# B&R Automation Studio project perfxxl (part 10)

#### pro_v.c
```c
#ifdef _DEFAULT_INCLUDES
	#include <AsDefault.h>
#endif
/*
                             *******************
******************************* C SOURCE FILE *******************************
**                           *******************                           **
**                                                                         **
** project  : BlueFin                                                      **
** filename : PRO_V.C                                                      **
** version  : 1.01                                                         **
** date     : 16.10.2008                                                   **
**                                                                         **
*****************************************************************************
** Abstract                                                                **
** ========                                                                **
**                                                                         **
** Copyright (c) 2008, Krause-Biagosch GmbH                                **
** All rights reserved.                                                    **
**                                                                         **
*****************************************************************************
VERSION HISTORY:
----------------
Version     : 1.00
Date        : 14.10.2008
Revised by  : Herbert Aden
Description : Original version

Version     : 1.01
Date        : 16.10.2008
Revised by  : Herbert Aden
Description : Pumps now only active, if machine is in ON mode

*/
#define _PRO_V_C_SRC

/****************************************************************************/
/**                                                                        **/
/**                           INCLUDE FILES                                **/
/**                                                                        **/
/****************************************************************************/

#include "glob_var.h"
#include "egmglob_var.h"
#include <math.h>

/****************************************************************************/
/**                                                                        **/
/**                       DEFINITIONS AND MACROS                           **/
/**                                                                        **/
/****************************************************************************/
/* NONE */

/****************************************************************************/
/**                                                                        **/
/**                      TYPEDEFS AND STRUCTURES                           **/
/**                                                                        **/
/****************************************************************************/
/* NONE */

/****************************************************************************/
/**                                                                        **/
/**                      PROTOTYPES OF LOCAL FUNCTIONS                     **/
/**                                                                        **/
/****************************************************************************/
/* NONE */

/****************************************************************************/
/**                                                                        **/
/**                      EXPORTED VARIABLES                                **/
/**                                                                        **/
/****************************************************************************/
/* NONE */

/****************************************************************************/
/**                                                                        **/
/**                           GLOBAL VARIABLES                             **/
/**                                                                        **/
/****************************************************************************/
/***
***/

/****************************************************************************/
/**                                                                        **/
/**                      TASK-LOCAL VARIABLES                              **/
/**                                                                        **/
/****************************************************************************/
_LOCAL    INT                 RefillStep;

/****************************************************************************/
/**                                                                        **/
/**                    MODULE-LOCAL VARIABLES                              **/
/**                                                                        **/
/****************************************************************************/
static    TON_10ms_typ        ReplPumpTimer;
static    TON_10ms_typ        CanisterFullTimer;
static    TOF_10ms_typ        CanisterNotFullTimer;

/****************************************************************************/
/**                                                                        **/
/**                      EXTERNAL VARIABLES                                **/
/**                                                                        **/
/****************************************************************************/

/****************************************************************************/
/**                                                                        **/
/**                          EXPORTED FUNCTIONS                            **/
/**                                                                        **/
/****************************************************************************/

void InitProV(void)
{
	RefillStep = 0;
	CanisterFullTimer.IN    = FALSE;
	CanisterNotFullTimer.IN = FALSE;
	ReplPumpTimer.IN = FALSE;
}

void ProV(void)
{

/*
 * Umwälzung immer, solange nicht leer (Levelswitch ist scließer!)
 */
	Out_DevCanister_Circulation =  In_DevCanister_Empty
								&& ControlVoltageOk
								&& EGMDeveloperTank.Enable;

	CanisterFullTimer.IN    = In_DevCanister_Full;
	CanisterNotFullTimer.IN = In_DevCanister_Full;
	CanisterFullTimer.PT = 1000;
	CanisterNotFullTimer.PT = 1000;
	TON_10ms(&CanisterFullTimer);
	TOF_10ms(&CanisterNotFullTimer);

	TON_10ms(&ReplPumpTimer);
/*
 * Befüllpumpe an für 1 min, wenn Levelschalter "voll" weggeht
 * Wenn Schalter wiederkommt, dann auf jeden Fall aus
 */

	if( !ControlVoltageOk
 	 || !EGMDeveloperTank.Enable
 	 )
 	{
 		RefillStep = 0;
 		ReplPumpTimer.IN = FALSE;
		Out_DevCanister_Replenish = FALSE;
 	}

	switch (RefillStep)
	{
		case 0:
		{
			if( !ControlVoltageOk
		 	 || !EGMDeveloperTank.Enable
		 	 )
		 		break;

		/* Pumpe an, Wartezeit 0,5 min triggern*/
			if(!CanisterNotFullTimer.Q)
			{
				ReplPumpTimer.IN = TRUE;
				ReplPumpTimer.PT = EGMAutoParam.PROV_PumpOnTime;
				Out_DevCanister_Replenish = TRUE;
				RefillStep = 10;
				break;
			}

			break;
		}
		case 10:
		{
		/* Wartezeit abgelaufen: Pumpe aus,nächster Schritt*/
			if(ReplPumpTimer.Q)
			{
				Out_DevCanister_Replenish = FALSE;
				ReplPumpTimer.IN = FALSE;
				RefillStep = 20;
				break;
			}
		/* Kanister wieder voll: Pumpe aus und fertig*/
			if(CanisterFullTimer.Q)
			{
				ReplPumpTimer.IN = FALSE;
				RefillStep = 0;
				Out_DevCanister_Replenish = FALSE;
				break;
			}

			break;
		}
		case 20:
		{
		/* Warten eine min */
			if(ReplPumpTimer.Q)
			{
				ReplPumpTimer.IN = FALSE;
				RefillStep = 0;
				break;
			}
			ReplPumpTimer.IN = TRUE;
			ReplPumpTimer.PT = EGMAutoParam.PROV_PumpOffTime; /* 5 min */
			break;
		}
	}

}
```

### Program Logical/Processor/egmauto (ANSIC, version 0.00.0)

#### auto.c
```c
#ifdef _DEFAULT_INCLUDES
	#include <AsDefault.h>
#endif
/*************************************************************************************************
 Handling of Automatic mode

*************************************************************************************************/

/****	Bedeutung der Ampel Signale

o = AUS, X = AN, b = blinkt

					Grün		Gelb		Rot
Aus					o			o			X
Aufheizen			o			o			X
Betriebsbereit		X			o			o
Verarbeitung		o			X			o
Reinigung			o			b			o
Störung				o			o			b
***/

/*********************************************************************************/
/*	Alarmliste */
/**
x	EGM_AlarmBitField[0]	AlarmNr 1	Notaus
x	EGM_AlarmBitField[1]	AlarmNr 2	kein Antriebstakt
x	EGM_AlarmBitField[2]	AlarmNr 3	EGMGummierung Füllstand zu niedrig
x	EGM_AlarmBitField[3]	AlarmNr 4	Vorspülen Füllstand zu niedrig
x	EGM_AlarmBitField[4]	AlarmNr 5	Nachspülen Füllstand zu niedrig
x	EGM_AlarmBitField[5]	AlarmNr 6	Entwickler Füllstand zu niedrig
x	EGM_AlarmBitField[6]	AlarmNr 7	Entwickler Temperatur zu niedrig
x	EGM_AlarmBitField[7]	AlarmNr 8	Entwickler Temperatur zu hoch
x	EGM_AlarmBitField[8]	AlarmNr 9	Nacherwärmung 1 Temperatur zu niedrig
x	EGM_AlarmBitField[9]	AlarmNr 10	Nacherwärmung 1 Temperatur zu hoch
x	EGM_AlarmBitField[10]	AlarmNr 11	Nacherwärmung 2 Temperatur zu niedrig
x	EGM_AlarmBitField[11]	AlarmNr 12	Nacherwärmung 2 Temperatur zu hoch
x	EGM_AlarmBitField[12]	AlarmNr 13	Plattenstau
	EGM_AlarmBitField[13]	AlarmNr 14	Entwickler zu alt
	EGM_AlarmBitField[14]	AlarmNr 15	E/A Modul nicht gefunden
x	EGM_AlarmBitField[15]	AlarmNr 16	Nacherw. Sensor 1 defekt
x	EGM_AlarmBitField[16]	AlarmNr 17	Nacherw. Sensor 2 defekt
x	EGM_AlarmBitField[17]	AlarmNr 18	Nacherw. Umgeb. Sensor defekt
x	EGM_AlarmBitField[18]	AlarmNr 19	Entwickler Temp. Sensor defekt
x	EGM_AlarmBitField[19]	AlarmNr 20	Nacherw. Heizung 1 defekt
x	EGM_AlarmBitField[20]	AlarmNr 21	Nacherw. Heizung 2 defekt
	EGM_AlarmBitField[21]	AlarmNr 22	Vorspülstation Befüllen fehlgeschlagen
	EGM_AlarmBitField[22]	AlarmNr 23	Nachspülstation Befüllen fehlgeschlagen
	EGM_AlarmBitField[23]	AlarmNr 24	Entwickler Befüllen fehlgeschlagen
x	EGM_AlarmBitField[24]	AlarmNr 25	Nacherwärmung 1 überhitzt
x	EGM_AlarmBitField[25]	AlarmNr 26	Nacherwärmung 2 überhitzt
x	EGM_AlarmBitField[26]	AlarmNr 27	Entwickler überhitzt
x	EGM_AlarmBitField[27]	AlarmNr 28	Antrieb: Geschwindigkeitsabweichung zu groß
x	EGM_AlarmBitField[28]	AlarmNr 29	Temperaturmodul nicht gefunden
**/

#include "EGMglob_var.h"
#include "glob_var.h"
#include "auxfunc.h"

#define MM_PER_PULSE (251.0/18.0)
#define NUMBER_OF_TIMING_CYCLES 10

#define LAMPTESTTIME 50 /*  *10 ms*/

_GLOBAL BOOL	Clock_1s;

R_TRIGtyp	RPMSignalEdgeR;

R_TRIGtyp	InputSensorEdgeR,OutputSensorEdgeR;
F_TRIGtyp	InputSensorEdgeF,OutputSensorEdgeF;
TON_10ms_typ	PlateInputTimer,StandbyDelay;
TON_10ms_typ	InputSensorOnDelay,OutputSensorOnDelay,ProcessingTimer;
TOF_10ms_typ	InputSensorOffDelay,OutputSensorOffDelay;

/*Timer für Spülprogramm*/
TON_10ms_typ	CleaningTimer;

BOOL AutoInit,OffInit,WaitForStandby;
_GLOBAL REAL PlateLength; /* wird in lccount berechnet */
_LOCAL	STRING CurrentPlateName[MAXPLATETYPENAME+6];
_LOCAL	INT PlatesInMachine,TimeAtPlateInput;
_LOCAL INT	DontCheckHeating;
REAL tmpval;
int i;
BOOL	 EnablePulseCounter;
_LOCAL BOOL	OnButton,OffButton;
_LOCAL UDINT CleaningTimerDisplay,CleaningTimerOverallDisplay;

_LOCAL UDINT	TEST;

/* Variable, die genauso lange true ist, wie der sensor Eingang, aber über  ein- und ausschaltverzögerung entprellt*/
_GLOBAL	BOOL PlateOverSensor;

/* Variablen für Ampelansteuerung, interne Merker, werden an zentraler Stelle auf die Ausgänge kopiert
wegen Lampentest Funktion*/
BOOL	InternalLightGreen;
BOOL	InternalLightRed;
BOOL	InternalLightYellow;
BOOL	FatalError;
_LOCAL BOOL TriggerLampTest;
TON_10ms_typ		HornTimer1,HornTimer2,LampTestTimer;
int LampTestStep,LampTestCycle,LampTestReturnStep;
TP_10ms_typ		BlinkTimer1,BlinkTimer2;

F_TRIGtyp ServiceKeyEdgeF;

R_TRIGtyp AlarmTrigger[EGM_MAXALARMS];
_GLOBAL BOOL	HornActive;

static    TON_10ms_typ        WaitForOutputTimer;
static	BOOL	OutputBlocked;

/**
	Bei allen Platten im FIFO die Position um Betrag X erhöhen
**/
void FIFOChangePlatePosition(REAL X)
{
	int i = 0;
	REAL BackEnd;
	do
	{
		if (EGMPlateFIFO[i].Used)
		{
			EGMPlateFIFO[i].Position += X;
			BackEnd = (EGMPlateFIFO[i].Position - EGMPlateFIFO[i].Length);
			/* Trigger Waiting for output
			 */
			if(  (EGMPlateFIFO[i].Position > ((MACHINELENGTH - 0.35) * 1000))
			  && (EGMPlateFIFO[i].Status != PS_OUTPUTREACHED)
			  )
				EGMPlateFIFO[i].Status = PS_WAITINGFOROUTPUT;

			if(  (BackEnd > ((MACHINELENGTH + 0.15) * 1000))
			  && (EGMPlateFIFO[i].Status == PS_OUTPUTREACHED)
			  )
			{
				OutputBlocked = TRUE;
			}
		}
		i++;
	}
	while (i <FIFOLENGTH);

}

/**
	Alle Platten im FIFO um 1 Platz weiterrücken
**/
void FIFOShift(void)
{
	int i = FIFOLENGTH-2;

	do
	{
		if (EGMPlateFIFO[i].Used)
		{
			EGMPlateFIFO[i+1] = EGMPlateFIFO[i];
		}
		i--;
	}
	while (i>=0);
	EGMPlateFIFO[0].Used = FALSE;
	EGMPlateFIFO[0].Position = 0;
	EGMPlateFIFO[0].Length =  0;
	EGMPlateFIFO[0].Status = PS_NONE;
}

/**
	FIFO mit Platten für die Darstellung bearbeiten
**/
void HandleFIFO()
{
	RPMSignalEdgeR.CLK = RPMCheck;
	R_TRIG(&RPMSignalEdgeR);
	if ((CurrentMode == M_AUTO)
	&& ((CurrentState==S_PROCESSING) || (CurrentState==S_STARTPROCESSING))
	)
	{
/* mit jedem Antriebspuls werden die Platten um einen festen Betrag X weitergefördert*/
		if(RPMSignalEdgeR.Q )
			FIFOChangePlatePosition(MM_PER_PULSE);

/* mit steigender Flanke eine neue Platte im FIFO erzeugen*/
		if(InputSensorEdgeR.Q)
		{
			EGMPlateFIFO[0].Used = TRUE;
			EGMPlateFIFO[0].Position = 0;
			EGMPlateFIFO[0].Length =  0;
			EGMPlateFIFO[0].Status = PS_RUNNING;
		}
/*wenn im FIFO eine Platte am Anfang steht und der Sensor belegt bleibt, wird diese länger*/
		if(PlateOverSensor)
		{
			if(RPMSignalEdgeR.Q )
				EGMPlateFIFO[0].Length += MM_PER_PULSE;
		}
/* mit fallender Flanke die Platte im FIFO weiterschieben*/
		if(InputSensorEdgeF.Q)
		{
			FIFOShift();
			if(EGMPlatesInFIFO < (FIFOLENGTH - 1) )
				EGMPlatesInFIFO++;
		}

/* mit steigender Flanke des Ausgangssensors den Status der letzten Platte im FIFO wechseln */
		if(OutputSensorEdgeR.Q)
		{
			if (EGMPlatesInFIFO > 0 && EGMPlatesInFIFO < FIFOLENGTH)
			{
				if(EGMPlateFIFO[EGMPlatesInFIFO].Status == PS_WAITINGFOROUTPUT)
					EGMPlateFIFO[EGMPlatesInFIFO].Status = PS_OUTPUTREACHED;
			}
		}

/* mit fallender Flanke des Ausgangssensors die letzte Platte im FIFO Löschen*/
		if(OutputSensorEdgeF.Q)
		{
			if(OutputBlocked)
				EGM_AlarmBitField[12] = 0;

			OutputBlocked = FALSE;
			if (EGMPlatesInFIFO > 0 && EGMPlatesInFIFO < FIFOLENGTH)
			{
				EGMPlateFIFO[EGMPlatesInFIFO].Used = FALSE;
				EGMPlateFIFO[EGMPlatesInFIFO].Position = 0;
				EGMPlateFIFO[EGMPlatesInFIFO].Length =  0;
				EGMPlateFIFO[EGMPlatesInFIFO].Status = PS_NONE;
				EGMPlatesInFIFO--;
			}
		}
/* Auslauf blockiert: warten, bis alle Platten raus sind, dann Fehlermeldung*/
		if(OutputBlocked)
		{
			int i;
			REAL BackEnd;
			for(i=FIFOLENGTH;i>0;i--)
			{
				if(EGMPlateFIFO[i].Used)
				{
					BackEnd = (EGMPlateFIFO[i].Position - EGMPlateFIFO[i].Length);
					if(BackEnd > ((MACHINELENGTH - 0.35) * 1000))
					{
						EGMPlateFIFO[i].Used = FALSE;
						EGMPlateFIFO[i].Position = 0;
						EGMPlateFIFO[i].Length =  0;
						EGMPlateFIFO[i].Status = PS_NONE;
						if(EGMPlatesInFIFO > 0)
							EGMPlatesInFIFO--;
						if(PlatesInMachine > 0)
							PlatesInMachine--;
					}
				}
			}
			if(EGMPlatesInFIFO == 0 && !EGM_AlarmBitField[12])
			{
				ShowMessage(104,138,0,CAUTION,OKONLY, FALSE);
				EGM_AlarmBitField[12] = 1;
			}
		}

	}
	else
	if (((CurrentMode == M_AUTO)&& (CurrentState == S_READY))
	|| (PlatesInMachine == 0)
	)
	{
		int i;
		EGMPlatesInFIFO = 0;
		for( i = 0; i < FIFOLENGTH; i++)
		{
			EGMPlateFIFO[i].Used = 0;
			EGMPlateFIFO[i].Position = 0;
			EGMPlateFIFO[i].Length =  0;
		}
	}
}

int	FindPlateType(UDINT parLength)
{
	int i;
	int Deviation,MinDeviation,PosInTable;
	BOOL	transverse;

	MinDeviation = 32000; /* Startwert: Abweichung riesig*/
	transverse = FALSE;
	for (i=1;i<MAXPLATETYPES;i++)
	{
		Deviation = abs(EGMPlateTypes[i].SizeX - parLength);
		if (Deviation < MinDeviation)
		{
			MinDeviation = Deviation;
			PosInTable = i;
			transverse = FALSE;
		}
/*
		Deviation = abs(EGMPlateTypes[i].SizeY - parLength);
		if (Deviation < MinDeviation)
		{
			MinDeviation = Deviation;
			PosInTable = i;
			transverse = TRUE;
		}
*/
	}
	if (transverse)
		return PosInTable+MAXPLATETYPES;
	else
		return PosInTable;
}

void LampAndHorn(void)
{
	int i,j,k;
/*
 * definiert die Alarme, die eine Meldung auf dem Hauptbild auslösen
 * -1 ist Ende Kennung der Liste!
 * Achtung: Bei Veränderung muss auch in pics.c "case 101" angepasst werden
 *          Alarmnummern um 1 versetzt zu Alarmnummer in Visu, zB AlarmNr 49 zeigt
 *          in Visu Alarmnummer 50 an!!
 */
	int MessageAlarms[]={0,2,12,33,34,35,36,37,38,39,40,-1};

/* ********************************************************************************/
/* Ampel */
/* ********************************************************************************/
	BlinkTimer1.PT = 30;
	BlinkTimer2.PT = 30;
	TON_10ms(&LampTestTimer);
	BlinkTimer1.IN = ! BlinkTimer2.Q;
	TP_10ms(&BlinkTimer1);
	BlinkTimer2.IN = ! BlinkTimer1.Q;
	TP_10ms(&BlinkTimer2);

	switch (LampTestStep)
	{
		case 0:
		{
			int i;
			BOOL flag;
			flag = 0;
			for (i=0;i<EGM_MAXALARMS;i++)
			{
/* EGMPreheat Temperatur zu niedrig nur relevant, wenn der Regler auch an ist*/
				if (i==8 || i==10)
					flag = flag || (EGM_AlarmBitField[i] && EGMPreheat.Enable && !DontCheckHeating);
				else
					flag = flag || EGM_AlarmBitField[i];
			}

/*solange kein Lampentest ist: interne Ampelmerker auf Ausgänge kopieren*/
			if (flag)
			{
				LightRed = BlinkTimer1.Q;
				LightGreen = 0;
				LightYellow = 0;
			}
			else
			{
				LightGreen = InternalLightGreen;
				LightYellow = InternalLightYellow;
				if (FatalError)
					LightRed = InternalLightRed && BlinkTimer1.Q;
				else
					LightRed = InternalLightRed;
			}

/* warten auf Trigger*/
			if (TriggerLampTest)
			{
				LampTestStep = 1;
				LampTestTimer.IN = 0;
				LampTestReturnStep = 0;
				Horn = 1;
			}
			break;
		}
		case 1:
		{
			LightGreen = 1;
			LightRed = 0;
			LightYellow = 0;
			LampTestStep = 100;
			LampTestReturnStep = 5;
			break;
		}
		case 5:
		{
			LightGreen = 0;
			LightRed = 0;
			LightYellow = 1;
			LampTestStep = 100;
			LampTestReturnStep = 10;
			break;
		}
		case 10:
		{
			LightGreen = 0;
			LightRed = 1;
			LightYellow = 0;
			LampTestStep = 100;
			LampTestReturnStep = 1;
			break;
		}
/*Warteschritt als Unterprogramm*/
		case 100:
		{
			if (!TriggerLampTest)
			{
				LampTestTimer.IN = 0;
				LampTestStep = 0;
				break;
			}

			LampTestTimer.IN = 1;
			LampTestTimer.PT = LAMPTESTTIME;
			if (LampTestTimer.Q)
			{
				LampTestTimer.IN = 0;
				LampTestStep = LampTestReturnStep;
			}
			break;
		}
	}

/* ********************************************************************************/
/*
 * Fehler, die einen Benutzereingriff erfordern, lösen die Hupe aus
 * z.B. Kanister leer, Gummierung leer
 * Hupe quittierbar im Hauptbild, kommt wieder, wenn ein Fehler neu
`* auftritt (Flanke)
 */
 	i = j = k = 0;

 	while (MessageAlarms[i] != -1)
 	{
 		j = MessageAlarms[i];
		AlarmTrigger[j].CLK = EGM_AlarmBitField[j];
		R_TRIG(&AlarmTrigger[j]);
/* wenn ein Alarm aus der Liste eine positive Flanke hat, dann Hupe an */
		if( AlarmTrigger[j].Q )
			HornActive = TRUE;
/* Wenn kein Alarm aus der Liste ansteht, wird k in keinem Durchlauf erhöht,
 * dann wird unten die Hupe ausgeschaltet
 */
		if( EGM_AlarmBitField[j] )
			k++;

		i++;
 	}
/* wenn alle Alarme der Liste 0 sind, dann wurde k nicht erhöht, dann Hupe aus; */
/* Hupe kann auch per Knopfdruck vom Bediener zurückgesetzt werden */
	if (k == 0)
		HornActive = FALSE;

	if (  HornActive
	  && !HornTimer2.Q )
		HornTimer1.IN = 1;
	else
		HornTimer1.IN = 0;

	HornTimer1.PT = 1000; /* alle 10 s*/
	TON_10ms(&HornTimer1);

	HornTimer2.PT = 200; /* 2 sec*/
	TON_10ms(&HornTimer2);

/* nach Zeit die Hupe ein */
	if (HornTimer1.Q  )
		HornTimer2.IN = 1;

	if (HornTimer2.Q)
		HornTimer2.IN = 0;
/* Hupe nur ansteuern wenn kein Lampentest*/
	if (LampTestStep == 0)
	{
/*
 * bei fatalem Fehler schneller Hup-Takt
 */
		if (FatalError)
			Horn = BlinkTimer1.Q;
		else
/*
 * bei "normalem" Fehler Hupe alle 10 sec für 2 sec an
 * wird oben getriggert, indem HornTimer1.IN gesetzt wird
 */
			Horn = HornTimer2.IN;
	}
/* ********************************************************************************/
}

_INIT void init()
{
	OutputBlocked = FALSE;
	FatalError  = 0;
	WaitForStandby = FALSE;
	CurrentMode = M_OFF;
	AutoInit = 1;
	CleaningTimer.IN = 0;
	CleaningTimer.PT = 100;
	SessionPlateCounter = 0;
	InternalLightGreen = 0;
	InternalLightYellow = 0;
	InternalLightRed = 0;
	Horn = 0;
	EGMPlatesInFIFO = 0;
	HornTimer1.IN = 0;
	HornTimer2.IN = 0;
	LampTestStep = 0;
	LampTestCycle = 0;
}

_CYCLIC void cyclic()
{
	EGM_AlarmBitField[14] =    (ModulStatus_PS  != 1)
							&& (ModulStatus_DI  != 1)
							&& (ModulStatus_DO1 != 1)
							&& (ModulStatus_DO2 != 1)
							&& (ModulStatus_DO3 != 1)
							&& (ModulStatus_AO  != 1)
							&& (ModulStatus_AT  != 1);
	if( !EGM_AlarmBitField[14])
	{
		EGM_AlarmBitField[28] = (ModulStatus_AT != 1);
		EGM_AlarmBitField[29] = (ModulStatus_DI != 1);
		EGM_AlarmBitField[30] = (ModulStatus_DO1 != 1) || (ModulStatus_DO2 != 1) || (ModulStatus_DO3 != 1);
		EGM_AlarmBitField[31] = (ModulStatus_AO != 1);
		EGM_AlarmBitField[32] = (ModulStatus_PS != 1);
	}
	else
	{
		EGM_AlarmBitField[28] = 0;
		EGM_AlarmBitField[29] = 0;
		EGM_AlarmBitField[30] = 0;
		EGM_AlarmBitField[31] = 0;
		EGM_AlarmBitField[32] = 0;
	}

	if (InputSensorEdgeR.Q)
		PlateOverSensor = TRUE;
	if (InputSensorEdgeF.Q)
		PlateOverSensor = FALSE;
	HandleFIFO();
	LampAndHorn();

/******************************************************/
/*
 * wenn die erste Platte im FIFO länger als 30 cm den Status WaitForOutput hat
 * dann ist das ein Plattenstau
 * Auswertung erfolgt im status Processing
 */
	WaitForOutputTimer.IN = (EGMPlateFIFO[EGMPlatesInFIFO].Status == PS_WAITINGFOROUTPUT)
	                        && !OutputBlocked;
/*	WaitForOutputTimer.PT = 1000;*/
/* 0,3 m -> 30 cm */
	WaitForOutputTimer.PT = (UDINT)
			(60.0 * 100.0 *
			(0.35 / ((REAL)EGMMainMotor.RatedRpm * EGMGlobalParam.MainMotorFactor)));
	TON_10ms(&WaitForOutputTimer);

/******************************************************/

/* aktuellen Status für die XML-Schnittstelle in Struktur eintragen */
	EGMState.mode = CurrentMode;
	EGMState.state = CurrentState;

/*Flankenerkennung aller Plattensensoren*/
	InputSensorEdgeR.CLK = InputSensorOnDelay.Q;
	InputSensorEdgeF.CLK = InputSensorOffDelay.Q;
	OutputSensorEdgeR.CLK = OutputSensorOnDelay.Q;
	OutputSensorEdgeF.CLK = OutputSensorOffDelay.Q;

	R_TRIG(&InputSensorEdgeR);
	R_TRIG(&OutputSensorEdgeR);
	F_TRIG(&InputSensorEdgeF);
	F_TRIG(&OutputSensorEdgeF);

	ServiceKeyEdgeF.CLK = ServiceKey;
	F_TRIG(&ServiceKeyEdgeF);
/* Timer für Spülprogramm*/
	TON_10ms(&CleaningTimer);
	CleaningTimerDisplay = (CleaningTimer.PT  - CleaningTimer.ET)/100;

/*Zeit messen, von steigender bis fallender Flanke*/
	PlateInputTimer.PT = 60000; /*soll nie erreicht werden*/
	TON_10ms(&PlateInputTimer);
	TON_10ms(&ProcessingTimer);
	TON_10ms(&StandbyDelay);
/*Entprellen je 1 sec*/
	InputSensorOnDelay.PT = 100;
	InputSensorOffDelay.PT = 100;
/*Entprellen je 1 sec*/
	OutputSensorOnDelay.PT = 100;
	OutputSensorOffDelay.PT = 100;
	InputSensorOnDelay.IN = InputSensor;
	InputSensorOffDelay.IN = InputSensor;
	OutputSensorOnDelay.IN = OutputSensor;
	OutputSensorOffDelay.IN = OutputSensor;
	TON_10ms(&InputSensorOnDelay);
	TON_10ms(&OutputSensorOnDelay);
	TOF_10ms(&InputSensorOffDelay);
	TOF_10ms(&OutputSensorOffDelay);
/*bei steigender Flanke starten*/
	if(InputSensorEdgeR.Q && !PlateInputTimer.IN)
	{
		PlateInputTimer.IN = 1;
	}
/*bei fallender Flanke stoppen*/
	if(InputSensorEdgeF.Q && PlateInputTimer.IN)
	{
		PlateInputTimer.IN = 0;
		TimeAtPlateInput = PlateInputTimer.ET;
	}

/* Bei Not Aus die Maschine in Stop setzen*/
	if (!ControlVoltageOk)
	{
		OffInit = 1;
		CurrentMode = M_OFF;
		CurrentState = S_OFF;
		InternalLightGreen = 0;
		InternalLightYellow = 0;
		InternalLightRed = Clock_1s;
	}
	EGM_AlarmBitField[0] = (!ControlVoltageOk);

/*****************************************************************/
/**  Signale an Belichter */
/*****************************************************************/
	if(  (CurrentMode == M_AUTO )
	  &&((CurrentState == S_READY) || (CurrentState == S_PROCESSING))
	  && !FatalError
	  && !PlateOverSensor
	  && (!EGMGum.LevelNotInRange || (!EGMGlobalParam.EnableGumSection && (MachineType==BLUEFIN_LOWCHEM)))
	  && ((EGMGum.PumpCmd == ON) || (!EGMGlobalParam.EnableGumSection && (MachineType==BLUEFIN_LOWCHEM)) )
	  && !OutputBlocked
	  )
	{
		Ready = 1;
		NoError = 1;
	}
	else
	{
		Ready = 0;
		if (FatalError || !ControlVoltageOk)
			NoError = 0;
		else
			NoError = 1;
	}
/*****************************************************************/
/*****************************************************************/

	switch (CurrentMode)
	{
		case M_OFF: /*OFF*/
		{
			FatalError = 0;
			EGM_AlarmBitField[12] = 0;
			OutputBlocked = FALSE;
			WaitForStandby = FALSE;
			PlatesInMachine = 0;
			CurrentState = S_OFF;
			EGMMainMotor.AutoRatedRpm = 0;
			EGMBrushMotor.AutoRatedRpm= 0;
			if (OffInit)
			{
				InternalLightGreen = 0;
				InternalLightYellow = 0;
				InternalLightRed = 1;

				EGMMainMotor.RatedRpm = 0;
				EGMBrushMotor.RatedRpm= 0;
/*Pumpen aus*/
				EGMGum.PumpCmd = OFF;
				if(MachineType == BLUEFIN_XS)
				{
					EGMPrewash.PumpCmd = OFF;
					if (EGMPrewashParam.ReplenishingMode == FRESHWATERONLY)
						EGMPrewash.Valve = CLOSE;

					EGMRinse.PumpCmd = OFF;
					if (EGMRinseParam.ReplenishingMode == FRESHWATERONLY)
						EGMRinse.Valve = CLOSE;
					EGMPrewash.Auto = 0;
					EGMRinse.Auto = 0;
				}
				Drying = OFF;
				EGMDeveloperTank.Enable = 0;
/*EGMPreheat Regelung aus und auf Manuell*/
				EGMPreheat.Enable = 0;
				for(i=0;i<4;i++)
					EGMPreheat.Auto[i] = 0;
				EGMDeveloperTank.Auto = 0;
/* V1.11 Gummierung Spülwasserventil AUS*/
				EGMGum.RinseValve = OFF;
			}

			EGMBrushMotor.Auto = 0;
			EGMMainMotor.Auto = 0;
			OffInit = 0;
			AutoInit =1;
			if (OnButton && ControlVoltageOk)
			{
				OnButton = 0;
				CurrentMode = M_AUTO;
			}
			break;
		}
		case M_AUTO:  /*AUTO*/
		{
			OffInit = 1;

			if (AutoInit)
			{
				InternalLightGreen = 0;
				InternalLightYellow = 0;
				InternalLightRed = 1;

				AutoInit = 0;
				EGMPreheatParam.RatedTemp[0] = EGMAutoParam.PreheatTemp;
				EGMPreheatParam.RatedTemp[1] = EGMAutoParam.PreheatTemp2;
				EGMPreheat.Enable = 1;
				for(i=0;i<4;i++)
					EGMPreheat.Auto[i] = 1;
				EGMDeveloperTankParam.RatedTemp = EGMAutoParam.DeveloperTemp;
				EGMDeveloperTank.Auto = 1;
				EGMBrushMotor.Auto = 1;
				EGMMainMotor.Auto = 1;
				EGMDeveloperTank.Enable = 1;
				if(MachineType == BLUEFIN_XS)
				{
					EGMPrewash.Auto = 1;
					EGMRinse.Auto = 1;
				}
				CurrentState = S_HEATING;

/* wenn Füllstand ok, dann die EGMGummierung-Zirkulationspumpe EIN*/
				if (!EGMGum.LevelNotInRange)
				{
					EGMGum.PumpCmd = ON;
					EGMGum.Auto = ON;
				}
				if(EGMGlobalParam.EnableGumSection || (MachineType == BLUEFIN_XS))
					EGMGum.Valve = ON;
			}

			if (OffButton )
			{
				OffButton = 0;
				if ((CurrentState == S_READY) || (CurrentState == S_HEATING) )
				{
					CurrentMode = M_INITCLEANING;
				}
				else
				if (CurrentState == S_PROCESSING )
				{
					CurrentState = S_WAITFORSTANDBY;
					WaitForStandby = 1;
				}
			}

			switch (CurrentState)
			{
				case S_HEATING:
				{
					BOOL LevelsOK;
					InternalLightYellow = 0;
					InternalLightGreen = 0;
					InternalLightRed = 1;

					EGMMainMotor.AutoRatedRpm = EGMAutoParam.StandbySpeed;
					EGMBrushMotor.AutoRatedRpm = EGMAutoParam.StandbyBrushSpeed;
					if(MachineType == BLUEFIN_XS)
					{
						LevelsOK = (!EGMPrewash.LevelNotInRange || (EGMPrewashParam.ReplenishingMode == FRESHWATERONLY))
		  			            && (!EGMRinse.LevelNotInRange   || (EGMRinseParam.ReplenishingMode == FRESHWATERONLY));
					}
					else
						LevelsOK = TRUE;

					if( ((EGMPreheat.TempInRange && EGMDeveloperTank.TempInRange) || DontCheckHeating)
	  				  &&  (!EGMGum.LevelNotInRange || (!EGMGlobalParam.EnableGumSection && (MachineType==BLUEFIN_LOWCHEM)))
	  				  &&   EGMDeveloperTank.LevelInRange
					  &&   LevelsOK
					  )
						CurrentState = S_READY;

					break;
				}
				case S_READY:
				{
					InternalLightGreen = 1;
					InternalLightRed = 0;
					InternalLightYellow = 0;

/*
 *2.08: bugfix, jetzt auch bei "ready"-> es erfolgt auch wieder
        Freigabe an Jet
 */
/* wenn Füllstand ok, dann die EGMGummierung-Zirkulationspumpe EIN*/
					if (!EGMGum.LevelNotInRange)
					{
						EGMGum.PumpCmd = ON;
						EGMGum.Auto = ON;
					}
					if(EGMGlobalParam.EnableGumSection || (MachineType == BLUEFIN_XS))
						EGMGum.Valve = ON;

					if (InputSensor)
					{
						CurrentState = S_STARTPROCESSING;
						break;
					}
					if(WaitForStandby)
					{
						WaitForStandby = 0;
						CleaningTimer.IN = 0;
						CurrentMode = M_INITCLEANING;
					}
					break;
				}
				case S_STARTPROCESSING:
				{
					EGMMainMotor.AutoRatedRpm = EGMAutoParam.Speed;
					EGMBrushMotor.AutoRatedRpm = EGMAutoParam.BrushSpeed;
/* Platte war 3 s im Einlauf: Verarbeitung läuft -> Schrittwechsel*/
					if (PlateInputTimer.ET > 300) /*3 s*/
					{
						PlatesInMachine = 0;
						CurrentState = S_PROCESSING;
						StandbyDelay.IN = 0;

						if(MachineType == BLUEFIN_XS)
						{
							if (EGMPrewashParam.ReplenishingMode != FRESHWATERONLY)
								EGMPrewash.PumpCmd = ON;
							else
								EGMPrewash.Valve = OPEN;

							if (EGMRinseParam.ReplenishingMode != FRESHWATERONLY)
								EGMRinse.PumpCmd = ON;
							else
								EGMRinse.Valve = OPEN;
						}
/* wenn Serviceschalter nicht umgelegt ist, Trocknung EIN */
						if (ServiceKey)
							Drying = ON;
					}
					else /* innerhalb der ersten 3s:*/
					{
					/*wenn Platte zu kurz im Einlauf: zurück*/
						if (InputSensorEdgeF.Q)
						{
							EGMMainMotor.AutoRatedRpm = EGMAutoParam.StandbySpeed;
							EGMBrushMotor.AutoRatedRpm = EGMAutoParam.StandbyBrushSpeed;
							CurrentState = S_READY;
							break;
						}
						else  /* nicht die negative Flanke vom Einlauf: abbruch, warten*/
							break;
					}
/***
das obligatorische break fehlt hier bewußt, da es vorher im if .. else eingebaut ist.
Wenn ein Start erkannt wird soll NICHT gebreakt werden, sondern direkt in PROCESSING
weitergemacht werden
***/
				}
				case S_WAITFORSTANDBY:
				case S_PROCESSING:
				{
					InternalLightGreen = 0;
					InternalLightYellow = 1;
					InternalLightRed = 0;
/* wenn Füllstände ok sind, dann die Zirkulationspumpen EIN*/
					if (!EGMGum.LevelNotInRange)
					{
						EGMGum.PumpCmd = ON;
						EGMGum.Auto = ON;
					}
					if(EGMGlobalParam.EnableGumSection || (MachineType == BLUEFIN_XS))
					EGMGum.Valve = ON;

					if(MachineType == BLUEFIN_XS)
					{
						if (!EGMPrewash.LevelNotInRange
						&& (!AlarmBitField[35])
						&& (EGMPrewashParam.ReplenishingMode != FRESHWATERONLY))
							EGMPrewash.PumpCmd = ON;

						if (!EGMRinse.LevelNotInRange
						&& (!AlarmBitField[36])
						&& (EGMRinseParam.ReplenishingMode != FRESHWATERONLY))
							EGMRinse.PumpCmd = ON;

	/* Prewash auf "Nur Frischwasser" -> Ventil Auf*/
						if (EGMPrewashParam.ReplenishingMode == FRESHWATERONLY)
							EGMPrewash.Valve = OPEN;

	/* Spülen auf "Nur Frischwasser" -> Ventil Auf*/
						if (EGMRinseParam.ReplenishingMode == FRESHWATERONLY)
							EGMRinse.Valve = OPEN;
					}
/* Überwachungstimer:
solange Platten in der Maschine sind, muß mindestens alle 2 min
der Auslaufsensor kommen
*/
					if (PlatesInMachine > 0)
					{
						if (OutputSensorEdgeR.Q)
							ProcessingTimer.IN = 0;
						else
						{
							ProcessingTimer.IN = 1;
							ProcessingTimer.PT = (UDINT)
								(60.0 * 100.0 *
								(MACHINELENGTH / ((REAL)EGMMainMotor.RatedRpm * EGMGlobalParam.MainMotorFactor)));

							/* Geschw > 1,5 m/min: 10 sec Sicherheit*/
							/* Geschw < 1,5 m/min: 20 sec Sicherheit*/
							if ( ((REAL)EGMMainMotor.RatedRpm * EGMGlobalParam.MainMotorFactor)<1.5 )
								ProcessingTimer.PT += 2000;
							else
								ProcessingTimer.PT += 1000;
						}
					}
					else /* PlatesInMachine is 0*/
					{
						ProcessingTimer.IN = 0;
						if( OutputSensorEdgeR.Q )
							PlatesInMachine = 1;
					}

/* Überwachungstimer schlägt an
 * -> ERROR
 */
					if( /* ProcessingTimer.Q
					 || */ WaitForOutputTimer.Q
					  )
					{
						CurrentState = S_ERROR;
						FatalError = 1;
						ProcessingTimer.IN = 0;
						ShowMessage(104,103,0,CAUTION,OKONLY, FALSE);

						EGM_AlarmBitField[12] = 1;
					}

/*wenn eine Platte den Ein- oder Auslaufsensor betätigt, dann  Trocknung EIN*/
					if ((InputSensor || OutputSensor) && ServiceKey)
						Drying = ON;
/* wenn Service Schalter umgelegt ist, wird die Trocknung immer Ausgeschaltet */
					if (ServiceKeyEdgeF.Q)
						Drying = OFF;

/*weitere Platten mitkriegen*/
					if (InputSensorEdgeF.Q)
					{
						int TypeNr;
						StandbyDelay.IN = 0;
						PlatesInMachine++;
						TypeNr = FindPlateType(PlateLength);
						if (TypeNr >= MAXPLATETYPES)
						{
							TypeNr -= MAXPLATETYPES;
							strcpy(CurrentPlateName,EGMPlateTypes[TypeNr].Name);
							strcat (CurrentPlateName," (q)");
						}
						else
							strcpy(CurrentPlateName,EGMPlateTypes[TypeNr].Name);

						OverallSqmCounter += EGMPlateTypes[TypeNr].Area;
						SessionSqmCounter += EGMPlateTypes[TypeNr].Area;
						ReplenishmentSqmCounter += EGMPlateTypes[TypeNr].Area;
						TopUpSqmCounter += EGMPlateTypes[TypeNr].Area;
						PrewashReplenishmentSqmCounter += EGMPlateTypes[TypeNr].Area;
						RinseReplenishmentSqmCounter += EGMPlateTypes[TypeNr].Area;
						SqmSinceDevChg += EGMPlateTypes[TypeNr].Area;

						ReplenishmentPlateCounter++;
						TopUpPlateCounter++;
						PrewashReplenishmentPlateCounter++;
						RinseReplenishmentPlateCounter++;
					}

/*auslaufende Platten mitkriegen*/
					if (OutputSensorEdgeF.Q )
					{
						PlatesInMachine--;
						OverallPlateCounter++;
						SessionPlateCounter++;
					}

					if (PlatesInMachine < 0) PlatesInMachine = 0;

					if ((PlatesInMachine == 0)	&& !InputSensor && !OutputSensor  )
					{
						StandbyDelay.IN = 1;
						StandbyDelay.PT = EGMAutoParam.StandbyDelay;
					}
					else
						StandbyDelay.IN = 0;

					if (StandbyDelay.Q)
					{
						StandbyDelay.IN = 0;
						EGMMainMotor.AutoRatedRpm = EGMAutoParam.StandbySpeed;
						EGMBrushMotor.AutoRatedRpm = EGMAutoParam.StandbyBrushSpeed;
						if(MachineType == BLUEFIN_XS)
						{
							if (EGMPrewashParam.ReplenishingMode == FRESHWATERONLY)
								EGMPrewash.Valve = CLOSE;
							if (EGMRinseParam.ReplenishingMode == FRESHWATERONLY)
								EGMRinse.Valve = CLOSE;

							EGMPrewash.PumpCmd = OFF;
							EGMRinse.PumpCmd = OFF;
						}
						Drying = OFF;
						CurrentState = S_READY;
					}

					break;
				}
				case S_ERROR:
				{
					InternalLightGreen = 0;
					InternalLightYellow = 0;
					InternalLightRed = 1;

					EGMMainMotor.RatedRpm = 0;
					EGMBrushMotor.RatedRpm= 0;
					EGMMainMotor.AutoRatedRpm = 0;
					EGMBrushMotor.AutoRatedRpm= 0;
	/*Pumpen aus*/
					EGMGum.PumpCmd = OFF;
					EGMGum.Auto = OFF;
					if(MachineType == BLUEFIN_XS)
					{
						EGMPrewash.PumpCmd = OFF;
						if (EGMPrewashParam.ReplenishingMode == FRESHWATERONLY)
							EGMPrewash.Valve = CLOSE;
						if (EGMRinseParam.ReplenishingMode == FRESHWATERONLY)
							EGMRinse.Valve = CLOSE;
						EGMRinse.PumpCmd = OFF;
					}
					Drying = OFF;
					EGMDeveloperTank.Enable = 0;
	/*EGMPreheat Regelung aus und auf Manuell*/
					EGMPreheat.Enable = 0;
					for(i=0;i<4;i++)
						EGMPreheat.Auto[i] = 0;
					EGMDeveloperTank.Auto = 0;
					if (AbfrageOK || AbfrageCancel)
					{
						FatalError = 0;
						CurrentState = S_OFF;
						CurrentMode = M_OFF;
						OffInit = 1;
						EGM_AlarmBitField[12] = 0;
					}
					break;
				}

/*****************************************************************************************************/
/*****************************************************************************************************/
/*****************************************************************************************************/
			}
			break;
		}
/*****************************************************************************************************/
		case M_INITCLEANING:
		{
			if((!EGMGlobalParam.EnableGumSection && (MachineType==BLUEFIN_LOWCHEM)))
			{
				FatalError = 0;
				CurrentState = S_OFF;
				CurrentMode = M_OFF;
				OffInit = 1;
				break;
			}

/* Funktionen für OFF schonmal vorweg nehmen: Heizungen aus, Bürsten aus */
			EGMBrushMotor.AutoRatedRpm= 0;
			EGMBrushMotor.RatedRpm= 0;
			EGMBrushMotor.Auto = 0;
			EGMDeveloperTank.Enable = 0;
/*EGMPreheat Regelung aus und auf Manuell*/
			EGMPreheat.Enable = 0;
			for(i=0;i<4;i++)
				EGMPreheat.Auto[i] = 0;
/*Entwicklertank Automatik aus*/
			EGMDeveloperTank.Auto = 0;

/* zum Start der Reinigung EGMGummierungspumpe aus, Ablaufventil auf Rückfluß in Behälter*/
			EGMGum.PumpCmd = OFF;
			EGMGum.Auto = OFF;
			EGMGum.Valve = ON;
/* Walzen auf Normalspeed*/
			EGMMainMotor.AutoRatedRpm = EGMAutoParam.Speed;
			CleaningTimer.IN = 1;
			CleaningTimer.PT = EGMAutoParam.WaitGumBackTime*100;
			CurrentMode = M_CLEANING;
			CurrentState = S_CLEANING1;
			CleaningTimerOverallDisplay = EGMAutoParam.WaitGumBackTime + EGMAutoParam.GumRinsingTime +
												EGMAutoParam.WaitGumRinseTime;
			break;
		}
		case M_CLEANING:
		{
			InternalLightYellow = Clock_1s;
			InternalLightRed = 0;
			InternalLightGreen = 0;

			CleaningTimerDisplay = (CleaningTimer.PT  - CleaningTimer.ET)/100;
/*Abbruch während des Reinigungszyklus*/
			if (OffButton)
			{
				OffButton = 0;
				EGMGum.PumpCmd = OFF;
				EGMGum.Auto = OFF;
/**/
				if (CurrentState == S_CLEANING1)
					EGMGum.Valve = ON;
				else
					EGMGum.Valve = OFF;
				EGMGum.RinseValve = OFF;
				CurrentMode = M_OFF;
				CurrentState = S_OFF;
				OffInit = 1;
				CleaningTimer.IN = 0;
				break;
			}

			switch (CurrentState)
			{
				case  S_CLEANING1:	/*warten, daß Gummierung zurückläuft*/
				{
					CleaningTimerOverallDisplay =  CleaningTimerDisplay + EGMAutoParam.GumRinsingTime +
												EGMAutoParam.WaitGumRinseTime;
					if (CleaningTimer.Q)
					{
						CleaningTimer.IN = 0;
						CurrentState = S_CLEANING2;
					}
					break;
				}
				case  S_CLEANING2:	/*Spülwasser an, Auslaß in Abfluß*/
				{
					CleaningTimerOverallDisplay =  CleaningTimerDisplay +
												EGMAutoParam.WaitGumRinseTime;
					if (EGMGum.RinseValve == ON)
					{
						CleaningTimer.IN = 1;
						CleaningTimer.PT = EGMAutoParam.GumRinsingTime*100;
					}
/* Spülwasser ein, Ablaufventil auf Ablauf in Abfluß*/
					EGMGum.RinseValve = ON;
					EGMGum.Valve = OFF;

					if (CleaningTimer.Q)
					{
/* Spülwasser aus, und warten, damit Spülwasser komplett in Abfluß fliessen kann*/
						EGMGum.RinseValve = OFF;
						CleaningTimer.IN = 0;
						CurrentState = S_CLEANING3;
					}
					break;
				}
				case  S_CLEANING3:	/*warten, daß Spülwasser komplett abgelaufen ist*/
				{
					CleaningTimerOverallDisplay = CleaningTimerDisplay;
					CleaningTimer.PT = EGMAutoParam.WaitGumRinseTime*100; /* 2 min*/
					CleaningTimer.IN = 1;

					if (CleaningTimer.Q)
					{
						CleaningTimer.IN = 0;
						CurrentState = S_OFF;
						CurrentMode = M_OFF;
						OffInit = 1;
						CleaningTimerDisplay = 0;
						CleaningTimerOverallDisplay = 0;
					}
					break;
				}

			}
			break;
		}
	}
/*in jedem Zyklus die Buttonmerker löschen*/
	OffButton=0;
	OnButton=0;
}
```

- auxfunc.h (reference to Logical/GlobalIncludes/auxfunc.h)

### Program Logical/Processor/egmser (ANSIC, version 0.00.0)

#### egmseriell.c
```c
#ifdef _DEFAULT_INCLUDES
	#include <AsDefault.h>
#endif
/****************************************************************************/
/*	serielle Kommunikation mit Thermo Kühl/Heizgerät                        */
/*	inklusive zyklisches Polling der Ist-Temperatur							*/
/*																			*/
/*	Versionsgeschichte:														*/
/*  Version		Datum		Änderung								von		*/
/*	1.0			05.02.07	erste Implementation					HA		*/
/*																			*/
/*																			*/
/****************************************************************************/
/* header files */
#include <dvframe.h>
#include <asstring.h>
#include <math.h>
#include <string.h>
#include <sys_lib.h>
#include "glob_var.h"
#include "egmglob_var.h"

#define THERMO_ADDRESS	(1)
#define READ_ACK		(0x00)
#define READ_STATUS 	(0x09)
#define READ_INT_TEMP	(0x20)
#define READ_EXT_TEMP	(0x21)
#define READ_SETPOINT	(0x70)
#define READ_LIMIT_LOW	(0x40)
#define READ_LIMIT_HIGH	(0x60)
#define READ_HEAT_P		(0x71)
#define READ_HEAT_I		(0x72)
#define READ_HEAT_D		(0x73)
#define READ_COOL_P		(0x74)
#define READ_COOL_I		(0x75)
#define READ_COOL_D		(0x76)

#define SET_SETPOINT	(0xF0)
#define SET_LIMIT_LOW	(0xC0)
#define SET_LIMIT_HIGH	(0xE0)
#define SET_HEAT_P		(0xF1)
#define SET_HEAT_I		(0xF2)
#define SET_HEAT_D		(0xF3)
#define SET_COOL_P		(0xF4)
#define SET_COOL_I		(0xF5)
#define SET_COOL_D		(0xF6)
#define ON_OFF_ARRAY	(0x81)

#define PRECISION_0_1_NOUNITS (0x10)
#define PRECISION_0_01_NOUNITS (0x20)
#define PRECISION_0_1_DEG_C (0x11)
#define PRECISION_0_01_DEG_C (0x21)

#define BIT0	((char)0x01)
#define BIT1	((char)0x02)
#define BIT2	((char)0x04)
#define BIT3	((char)0x08)
#define BIT4	((char)0x10)
#define BIT5	((char)0x20)
#define BIT6	((char)0x40)
#define BIT7	((char)0x80)

#define ANSWER_OK				(0)
#define ANSWER_INVALID			(-1)
#define ANSWER_BAD_CHECKSUM		(-2)
#define ANSWER_BAD_COMMAND		(-3)
#define ANSWER_INVALID_CHECKSUM	(-4)

#define HIGHBYTE(V)	((USINT) ((V>>8) & 0x00ff))
#define LOWBYTE(V)	((USINT) (V & 0x00ff))

/* variable declaration */
FRM_xopen_typ FrameXOpenStruct; 					/* variable of type FRMXOPEN */
FRM_close_typ FrameCloseStruct; 					/* variable of type FRMCLOSE */
XOPENCONFIG XOpenConfigStruct; 						/* variable of type XOPENCONFIG */
FRM_gbuf_typ FrameGetBufferStruct; 					/* variable of type FRMGBUF */
FRM_rbuf_typ FrameReleaseBufferStruct; 				/* variable of type FRMRBUF */
FRM_robuf_typ FrameReleaseOutputBufferStruct; 		/* variable of type FRMROBUF */
FRM_write_typ FrameWriteStruct; 					/* variable of type FRMWRITE */
FRM_read_typ FrameReadStruct; 						/* variable of type FRMREAD */
USINT Error, xopenOK;
USINT StringDevice[30], StringMode[30]; 			/* initialize strings for FRM_xopen */
USINT RequestData[READDATALENGTH]; /* array for requested Data */

_LOCAL BOOL StopPolling;
_LOCAL USINT PollingStep;
_LOCAL USINT RequestStep;
_LOCAL USINT timeout;

_LOCAL	USINT	ResendCounter;
_LOCAL	USINT	ErrorCounter;

_LOCAL	REAL	testval;

_GLOBAL	RTCtime_typ	RTCtime;
		USINT	lastSecond,SecondCounter;

_LOCAL UINT	Cooler_UnitOnInv;
_LOCAL UINT	Cooler_UnitStoppingInv;
_LOCAL UINT	Cooler_UnitFaultedInv;
_LOCAL UINT	Cooler_HTCFaultInv;
_LOCAL UINT	Cooler_PumpOnInv;
_LOCAL UINT	Cooler_CompressorOnInv;
_LOCAL UINT	Cooler_HeaterOnInv;
_LOCAL UINT	Cooler_LevelWarnInv;
_LOCAL UINT	Cooler_LevelFaultInv;
_LOCAL UINT	Cooler_LowTempWarnInv;
_LOCAL UINT	Cooler_HighTempWarnInv;
_LOCAL UINT	Cooler_LowTempFaultInv;
_LOCAL UINT	Cooler_HighTempFaultInv;
_LOCAL UINT	Cooler_RefrigTempHighInv;

static int Counter;
static int SendWaitCounter;
static int CurrentReadCommand,CurrentSetCommand;
static INT tmpval, SetPointOnly;

static int ReadCommands[] = {READ_STATUS, READ_INT_TEMP, READ_EXT_TEMP, READ_SETPOINT,
                             READ_LIMIT_LOW, READ_LIMIT_HIGH,
                             READ_HEAT_P, READ_HEAT_I, READ_HEAT_D,
                             READ_COOL_P, READ_COOL_I, READ_COOL_D };

static int SetCommands[] = {SET_SETPOINT,
                             SET_LIMIT_LOW, SET_LIMIT_HIGH,
                             SET_HEAT_P, SET_HEAT_I, SET_HEAT_D,
                             SET_COOL_P, SET_COOL_I, SET_COOL_D };

_LOCAL USINT StartUnit,StopUnit,ApplySetpoint;
static TON_10ms_typ	SetpointChangeTimer,SetpointChangeTimer2;
static BOOL SetpointChangeFlag;

/*------------------------------------------------------------------------------------
 initialize program starts here
-------------------------------------------------------------------------------------*/
_INIT void InitProgram(void)
{
	Cooler.NewValues.SetPoint = 22;
	Cooler.NewValues.LimitLow = 1.5;
	Cooler.NewValues.LimitHigh = 82;
	Cooler.NewValues.HeatP = 0.6;
	Cooler.NewValues.HeatI = 0.6;
	Cooler.NewValues.HeatD = 0.0;
	Cooler.NewValues.CoolP = 0.6;
	Cooler.NewValues.CoolI = 0.6;
	Cooler.NewValues.CoolD = 0.0;

	CurrentReadCommand = 0;
	CurrentSetCommand = 0;
	SetPointOnly = FALSE;
	lastSecond = 0;
	SecondCounter = 0;
	SendWaitCounter=0;
	Counter = 0;
	StopPolling = 0;
	ResendCounter = 0;
	ErrorCounter = 0;
	xopenOK = 0;
	strcpy(StringDevice, "IF1"); 							/* interface #1 */
	strcpy(StringMode, "/BD=19200 /PA=N /DB=8 /SB=1"); 		/* RS232 interface, 57600 BAUD, no parity, 8 data bits, 1 stop bit */

	/* initialize config structure */
	XOpenConfigStruct.idle = 6;                           /* in Zeichenlängen*/
	XOpenConfigStruct.delimc = 0;		/* keine Frame Ende Zeichen */
	XOpenConfigStruct.delim[0] = 10;	/* nicht benutzt, weil delimc==0 */
	XOpenConfigStruct.delim[1] = 13;	/* nicht benutzt, weil delimc==0 */
	XOpenConfigStruct.tx_cnt = 2;
	XOpenConfigStruct.rx_cnt = 2;
	XOpenConfigStruct.tx_len = 32;
	XOpenConfigStruct.rx_len = 32;
	XOpenConfigStruct.argc = 0;
	XOpenConfigStruct.argv = 0;

	/* initialize open structure */
	FrameXOpenStruct.enable = 1;
	FrameXOpenStruct.device = (UDINT) StringDevice;
	FrameXOpenStruct.mode = (UDINT) StringMode;
	FrameXOpenStruct.config = (UDINT) &XOpenConfigStruct;

	FRM_xopen(&FrameXOpenStruct); 						/* open an interface */

	if (FrameXOpenStruct.status == 0) 					/* check status */
	{
		xopenOK = 1;									/* set error level for FRM_xopen */

		/* initialize get buffer structure */
		FrameGetBufferStruct.enable = 1;
		FrameGetBufferStruct.ident = FrameXOpenStruct.ident;				/* get ident */

		/* initialize write structure */
		FrameWriteStruct.enable = 1;
		FrameWriteStruct.ident  = FrameXOpenStruct.ident;					/* get ident */

		/* initialize release output buffer structure */
		FrameReleaseOutputBufferStruct.enable = 1;
		FrameReleaseOutputBufferStruct.ident = FrameXOpenStruct.ident;		/* get ident */

		/* initialize read structure */
		FrameReadStruct.enable = 1;
		FrameReadStruct.ident = FrameXOpenStruct.ident;						/* get ident */

		/* initialize release buffer structure */
		FrameReleaseBufferStruct.enable = 1;
		FrameReleaseBufferStruct.ident = FrameXOpenStruct.ident;			/* get ident */

		/* initialize close structure */
		FrameCloseStruct.enable = 1;
		FrameCloseStruct.ident = FrameXOpenStruct.ident;					/* get ident */
	}
	else
	{
		xopenOK = 0;
	}
}

USINT CreateChecksum(char *buf, int length)
{
	int i,sum;

	sum = 0;
/* start at index 1 to leave out leading 0xCA */
	for(i=1;i<=length;i++)
	{
		sum += buf[i];
	}
	return  ~((USINT)sum);
}

int CreateCommand(char *cmdstring, INT Addr, USINT command, INT Value)
{
	int retval=0;

	cmdstring[0] = 0xCA;	/* Start cmd RS232 always $CA */
	cmdstring[1] = 0x00;	/* Addr MSB always 0 */
	if ( Addr <= 64 )
		cmdstring[2] = (USINT) Addr;
	else
		cmdstring[2] = 1;

	cmdstring[3] = command;		 	/* command  */

	switch (command)
	{
		case READ_STATUS:
		case READ_INT_TEMP:
		case READ_EXT_TEMP:
		case READ_SETPOINT:
		case READ_LIMIT_LOW:
		case READ_LIMIT_HIGH:
		case READ_HEAT_P:
		case READ_HEAT_I:
		case READ_HEAT_D:
		case READ_COOL_P:
		case READ_COOL_I:
		case READ_COOL_D:
		{
			cmdstring[4] = 0x00;			/* number of data bytes */
/* calculate checksum */
			cmdstring[5] = CreateChecksum(cmdstring,4);
/* length of command w/out data is always 6 bytes */
			retval = 6;
			break;
		}
		case SET_SETPOINT:
		case SET_LIMIT_LOW:
		case SET_LIMIT_HIGH:
		case SET_HEAT_P:
		case SET_HEAT_I:
		case SET_HEAT_D:
		case SET_COOL_P:
		case SET_COOL_I:
		case SET_COOL_D:
		{
			cmdstring[4] = 0x02;			/* number of data bytes */

			cmdstring[5] = HIGHBYTE(Value);
			cmdstring[6] = LOWBYTE(Value);
/* calculate checksum */
			cmdstring[7] = CreateChecksum(cmdstring,6);
/* length of command with data is always 8 bytes */
			retval = 8;
			break;
		}
		case ON_OFF_ARRAY:
		{
			cmdstring[4] = 0x08;			/* number of data bytes */
			if (Value == 1)
				cmdstring[5] = 0x01; /* Unit ON */
			else
			if (Value == 0)
				cmdstring[5] = 0x00; /* Unit OFF */

			cmdstring[6] = 0x02;
			cmdstring[7] = 0x02;
			cmdstring[8] = 0x02;
			cmdstring[9] = 0x02;
			cmdstring[10] = 0x00; /* 0.01 °C enable OFF */
			cmdstring[11] = 0x02;
			cmdstring[12] = 0x02;
/* calculate checksum */
			cmdstring[13] = CreateChecksum(cmdstring,12);
/* length of command with data is always 8 bytes */
			retval = 14;
			break;
		}
	}

	return retval;
}

SINT ParseAnswer(USINT *buf, INT Addr, INT length, USINT command, REAL *value)
{
	BOOL retval = ANSWER_INVALID;
	USINT qualifier;

	if( buf[0] != 0xCA
	 || buf[1] != 0
	 || buf[2] != (USINT) Addr
	  )
	  return ANSWER_INVALID;

	if(buf[3] == 0x0F)
	{
		switch (buf[5])
		{
			case 1: /* bad coommand */
			{
				retval = ANSWER_BAD_COMMAND;
				break;
			}
			case 3:/* bad checksum */
			{
				retval = ANSWER_BAD_CHECKSUM;
				break;
			}
			default: /* other cases not possible per definition*/
			{
				retval = ANSWER_INVALID;
				break;
			}
		}
		return retval;
	}
	else
	if(buf[3] != command)
		return ANSWER_INVALID;

	if( buf[4] <= 8)   /* max 8 data bytes allowed */
	{
/* Telegramm ok, auswerten */
		switch (command)
		{
			case READ_INT_TEMP:
			case READ_EXT_TEMP:
			case READ_SETPOINT:
			case READ_LIMIT_LOW:
			case READ_LIMIT_HIGH:
			case READ_HEAT_P:
			case READ_HEAT_I:
			case READ_HEAT_D:
			case READ_COOL_P:
			case READ_COOL_I:
			case READ_COOL_D:
			case SET_SETPOINT:
			case SET_LIMIT_LOW:
			case SET_LIMIT_HIGH:
			case SET_HEAT_P:
			case SET_HEAT_I:
			case SET_HEAT_D:
			case SET_COOL_P:
			case SET_COOL_I:
			case SET_COOL_D:
			{
				if( buf[4] == 3)
				{
					qualifier = buf[5];
		/* Wert aus Antwort isolieren und umrechnen */
					*value = buf[6]*256 + buf[7];
					if( qualifier == PRECISION_0_1_NOUNITS || qualifier == PRECISION_0_1_DEG_C)
						*value /= 10.0;
					else
					if( qualifier == PRECISION_0_01_NOUNITS || qualifier == PRECISION_0_01_DEG_C)
						*value /= 100.0;

					retval = ANSWER_OK;
				}
				else
					retval = ANSWER_INVALID;
				break;
			}
			case READ_STATUS:
			{
				if (buf[4] == 5)
				{
					Cooler.RawDataB1 = buf[5];
					Cooler.RawDataB2 = buf[6];
					Cooler.RawDataB3 = buf[7];
					Cooler.RawDataB4 = buf[8];
					Cooler.RawDataB5 = buf[9];

					Cooler.RTD1OpenFault         = (Cooler.RawDataB1 & BIT7) != 0;
					Cooler.RTD1ShortedFault      = (Cooler.RawDataB1 & BIT6) != 0;
					Cooler.RTD1Open              = (Cooler.RawDataB1 & BIT5) != 0;
					Cooler.RTD1Shorted           = (Cooler.RawDataB1 & BIT4) != 0;
					Cooler.RTD3OpenFault         = (Cooler.RawDataB1 & BIT3) != 0;
					Cooler.RTD3ShortedFault      = (Cooler.RawDataB1 & BIT2) != 0;
					Cooler.RTD3Open              = (Cooler.RawDataB1 & BIT1) != 0;
					Cooler.RTD3Shorted           = (Cooler.RawDataB1 & BIT0) != 0;

					Cooler.RTD2OpenFault         = (Cooler.RawDataB2 & BIT7) != 0;
					Cooler.RTD2ShortedFault      = (Cooler.RawDataB2 & BIT6) != 0;
					Cooler.RTD2OpenWarn          = (Cooler.RawDataB2 & BIT5) != 0;
					Cooler.RTD2ShortedWarn       = (Cooler.RawDataB2 & BIT4) != 0;
					Cooler.RTD2Open              = (Cooler.RawDataB2 & BIT3) != 0;
					Cooler.RTD2Shorted           = (Cooler.RawDataB2 & BIT2) != 0;
					Cooler.RefrigHighTemp        = (Cooler.RawDataB2 & BIT1) != 0;
					Cooler.HTCFault              = (Cooler.RawDataB2 & BIT0) != 0;

					Cooler.HighFixedTempFault    = (Cooler.RawDataB3 & BIT7) != 0;
					Cooler.LowFixedTempFault     = (Cooler.RawDataB3 & BIT6) != 0;
					Cooler.HighTempFault         = (Cooler.RawDataB3 & BIT5) != 0;
					Cooler.LowTempFault          = (Cooler.RawDataB3 & BIT4) != 0;
					Cooler.LowLevelFault         = (Cooler.RawDataB3 & BIT3) != 0;
					Cooler.HighTempWarn          = (Cooler.RawDataB3 & BIT2) != 0;
					Cooler.LowTempWarn           = (Cooler.RawDataB3 & BIT1) != 0;
					Cooler.LowLevelWarn          = (Cooler.RawDataB3 & BIT0) != 0;

					Cooler.BuzzerOn              = (Cooler.RawDataB4 & BIT7) != 0;
					Cooler.AlarmMuted            = (Cooler.RawDataB4 & BIT6) != 0;
					Cooler.UnitFaulted           = (Cooler.RawDataB4 & BIT5) != 0;
					Cooler.UnitStopping          = (Cooler.RawDataB4 & BIT4) != 0;
					Cooler.UnitOn                = (Cooler.RawDataB4 & BIT3) != 0;
					Cooler.PumpOn                = (Cooler.RawDataB4 & BIT2) != 0;
					Cooler.CompressorOn          = (Cooler.RawDataB4 & BIT1) != 0;
					Cooler.HeaterOn              = (Cooler.RawDataB4 & BIT0) != 0;

					Cooler.RTD2Controlling       = (Cooler.RawDataB5 & BIT7) != 0;
					Cooler.HeatLEDFlashing       = (Cooler.RawDataB5 & BIT6) != 0;
					Cooler.CoolLEDFlashing       = (Cooler.RawDataB5 & BIT5) != 0;
					Cooler.CoolLEDOn             = (Cooler.RawDataB5 & BIT4) != 0;

					retval = ANSWER_OK;
				}
				else
					retval = ANSWER_INVALID;
				break;
			}
		}
	}
	else	/* number of data bytes not valid (>8) */
		retval = ANSWER_INVALID;

	return retval;
}

/*--------------------------------------------------------------------------------------
 cyclic program start here
--------------------------------------------------------------------------------------*/
_CYCLIC void CyclicProgram(void)
{
	Cooler_UnitOnInv              = !Cooler.UnitOn;
	Cooler_UnitStoppingInv        = !Cooler.UnitStopping;
	Cooler_UnitFaultedInv         = !Cooler.UnitFaulted;
	Cooler_PumpOnInv              = !Cooler.PumpOn;
	Cooler_CompressorOnInv        = !Cooler.CompressorOn;
	Cooler_HeaterOnInv            = !Cooler.HeaterOn;
	Cooler_LevelWarnInv           = !Cooler.LowLevelWarn;
	Cooler_LevelFaultInv          = !Cooler.LowLevelFault;
	Cooler_LowTempWarnInv         = !Cooler.LowTempWarn;
	Cooler_HighTempWarnInv        = !Cooler.HighTempWarn;
	Cooler_LowTempFaultInv        = !Cooler.LowTempFault;
	Cooler_HighTempFaultInv       = !Cooler.HighTempFault;
	Cooler_RefrigTempHighInv      = !Cooler.RefrigHighTemp;
	Cooler_HTCFaultInv            = !Cooler.HTCFault;

/*
 * if New setpoint and current Setpoint differ less than 3 °C but are not equal,
 * then we send the new setpoint because it will not be sent automatically due
 * to if(diff>3) clause
 */
	TON_10ms(&SetpointChangeTimer);
	TON_10ms(&SetpointChangeTimer2);

	SetpointChangeTimer.PT = 6000; /* 1 min */
	if( (fabs(Cooler.CurrentValues.SetPoint-Cooler.NewValues.SetPoint) < 3.0)
	&&  (fabs(Cooler.CurrentValues.SetPoint-Cooler.NewValues.SetPoint) > 0.2)
	&&  !SetpointChangeTimer.Q
	 )
		SetpointChangeTimer.IN = TRUE;
	else
		SetpointChangeTimer.IN = FALSE;

/*
 * more than 3 °C diff for more than 20 sec: apply new setpoint
 */
	TON_10ms(&SetpointChangeTimer2);
	SetpointChangeTimer2.PT = 2000; /* 20 sec */
	if( (fabs(Cooler.CurrentValues.SetPoint-Cooler.NewValues.SetPoint) > 3.0)
	&&  !SetpointChangeTimer2.Q
	 )
		SetpointChangeTimer2.IN = TRUE;
	else
		SetpointChangeTimer2.IN = FALSE;

	if(SetpointChangeTimer.Q || SetpointChangeTimer2.Q)
		SetpointChangeFlag = TRUE;

	if (xopenOK == 1)
	{

/******************************************************************/
/* Cyclic polling of current Temperature and status */
/******************************************************************/

		switch (PollingStep)
		{
			case 0:
			{
			/*
			 * Start command from Developertank task
			 */
				if( Cooler.Cmd_Start )
					StartUnit = TRUE;

				if (StartUnit)
				{
					Cooler.Cmd_Start = FALSE;
					PollingStep = 10;
	 				ResendCounter = 0;
					break;
				}
			/*
			 * Stop command from Developertank task
			 */
				if( Cooler.Cmd_Stop )
					StopUnit = TRUE;

				if (StopUnit)
				{
					Cooler.Cmd_Stop = FALSE;
					PollingStep = 10;
	 				ResendCounter = 0;
					break;
				}

				if (ApplySetpoint	/* button */
				|| (SetpointChangeFlag) /* flag from timer */
				)
				{
					if(!ApplySetpoint) /*not the button, but SetPoint changed by Application */
						SetPointOnly = TRUE;
					else
						SetPointOnly = FALSE;

					SetpointChangeFlag = FALSE;
					PollingStep = 20;
					ApplySetpoint = 0;
	 				ResendCounter = 0;
	 				CurrentSetCommand = 0;
					break;
				}

/* every 1 sec */
				if( RTCtime.second != lastSecond)
				{
					if(SecondCounter >= 1 )
					{
						PollingStep++;
						ResendCounter = 0;
						SecondCounter = 0;
					}
					else
						SecondCounter++;
					lastSecond = RTCtime.second;
					break;
				}

				break;
			}
/* 1st Step: send the GET Temp command */
			case 1:
			{
				FRM_gbuf(&FrameGetBufferStruct); 				/* get send buffer */

				if (FrameGetBufferStruct.status == 0) 			/* check status */
				{
					int length;

					length = CreateCommand((USINT*)FrameGetBufferStruct.buffer,
					                        THERMO_ADDRESS, ReadCommands[CurrentReadCommand], 0);
					/* initialize write structure */
					FrameWriteStruct.buffer = FrameGetBufferStruct.buffer;		/* get adress of send buffer */
					FrameWriteStruct.buflng = length;

					FRM_write(&FrameWriteStruct); 				/* write data to interface */

					if (FrameWriteStruct.status != 0) 			/* check status */
					{
						/* initialize release output buffer structure */
						FrameReleaseOutputBufferStruct.buffer = FrameGetBufferStruct.buffer;
						FrameReleaseOutputBufferStruct.buflng = FrameGetBufferStruct.buflng;
						FRM_robuf(&FrameReleaseOutputBufferStruct); 	/* release output buffer */

						Error = 3; 					/* set error level for FRM_write */

						if (FrameReleaseOutputBufferStruct.status != 0) 		/* check status */
						{
							Error = 4; 				/* set error level for FRM_robuf */
						}
					}
				}
	/*TODO: Fehler auswerten wenn getBuffer fehlschlägt (8071)*/
				PollingStep++;
				timeout = 0;
				break;
			}
/* wait for the answer */
			case 2:
			{
				/* initialize read structure */
				FRM_read(&FrameReadStruct); 						/* read data from interface */

				if (FrameReadStruct.status == 0) 					/* check status */
				{
					/* Checksum ok? */
					USINT tmp = CreateChecksum((USINT *)FrameReadStruct.buffer,FrameReadStruct.buflng-2);

					if( tmp == ((USINT *)FrameReadStruct.buffer)[FrameReadStruct.buflng-1] )
					{
						/* checksum OK */
						if(ParseAnswer((USINT *)FrameReadStruct.buffer, THERMO_ADDRESS,
						            FrameReadStruct.buflng, ReadCommands[CurrentReadCommand], &testval) != 0)
						{
							Error = 12; /* answer not correct*/
						}
						else	/* Answer formal OK */
						{
							/* Answer formal OK, value in testval */
							switch (ReadCommands[CurrentReadCommand])
							{
								case READ_STATUS: break;/* status is put into struct direcrly in parser */
								case READ_INT_TEMP:
								{
									Cooler.IntTemp = testval;
									break;
								}
								case READ_EXT_TEMP:
								{
									Cooler.ExtTemp = testval;
									break;
								}
								case READ_SETPOINT:
								{
									Cooler.CurrentValues.SetPoint = testval;
									break;
								}
								case READ_LIMIT_LOW:
								{
									Cooler.CurrentValues.LimitLow = testval;
									break;
								}
								case READ_LIMIT_HIGH:
								{
									Cooler.CurrentValues.LimitHigh = testval;
									break;
								}
								case READ_HEAT_P:
								{
									Cooler.CurrentValues.HeatP = testval;
									break;
								}
								case READ_HEAT_I:
								{
									Cooler.CurrentValues.HeatI = testval;
									break;
								}
								case READ_HEAT_D:
								{
									Cooler.CurrentValues.HeatD = testval;
									break;
								}
								case READ_COOL_P:
								{
									Cooler.CurrentValues.CoolP = testval;
									break;
								}
								case READ_COOL_I:
								{
									Cooler.CurrentValues.CoolI = testval;
									break;
								}
								case READ_COOL_D:
								{
									Cooler.CurrentValues.CoolD = testval;
									break;
								}
							}
						}

					}
					else
					{
						/* checksum error */
						Error = 11;
					}

					/* initialize release buffer structure */
					FrameReleaseBufferStruct.buffer = FrameReadStruct.buffer;	/* get adress of read buffer */
					FrameReleaseBufferStruct.buflng = FrameReadStruct.buflng; 	/* get length of read buffer */

					FRM_rbuf(&FrameReleaseBufferStruct); 			/* release read buffer */

					ResendCounter = 0;

					if (FrameReleaseBufferStruct.status != 0) 				/* check status */
					{
						Error = 6; 					/* set error level for FRM_rbuf */
					}
					if (CurrentReadCommand < 11)
					{
						CurrentReadCommand++;
						PollingStep = 1;
					}
					else
					{
						CurrentReadCommand = 0;
						PollingStep = 0;
					}
				}
				else
				{
					Error = 5; 						/* set error level for FRM_read */
					timeout++;
					if (timeout >= 20) /* 20*cyclic (->2s) time no answer */
					{
						if(ResendCounter >= 5) /*5 times tried? -> error*/
						{
							if (CurrentReadCommand < 11)
							{
								CurrentReadCommand++;
								PollingStep = 1;
							}
							else
							{
								CurrentReadCommand = 0;
								PollingStep = 0;
							}
							ResendCounter = 0;
						}
						else
						{
							ErrorCounter++;
							ResendCounter++;
							PollingStep = 1;
						}
					}
				}
				break;
			}

/*********************************************************************************************/
/*********************************************************************************************/
/*********************************************************************************************/
/*  send the Start Unit command */
			case 10:
			{
				FRM_gbuf(&FrameGetBufferStruct); 				/* get send buffer */

				if (FrameGetBufferStruct.status == 0) 			/* check status */
				{
					int length;

					if (StartUnit)
					{
						length = CreateCommand((USINT*)FrameGetBufferStruct.buffer,
					                        THERMO_ADDRESS, ON_OFF_ARRAY, 1 );
					    StartUnit = 0;
					}
					else
					if (StopUnit)
					{
						length = CreateCommand((USINT*)FrameGetBufferStruct.buffer,
					                        THERMO_ADDRESS, ON_OFF_ARRAY, 0 );
					    StopUnit = 0;
					}

					/* initialize write structure */
					FrameWriteStruct.buffer = FrameGetBufferStruct.buffer;		/* get adress of send buffer */
					FrameWriteStruct.buflng = length;

					FRM_write(&FrameWriteStruct); 				/* write data to interface */

					if (FrameWriteStruct.status != 0) 			/* check status */
					{
						/* initialize release output buffer structure */
						FrameReleaseOutputBufferStruct.buffer = FrameGetBufferStruct.buffer;
						FrameReleaseOutputBufferStruct.buflng = FrameGetBufferStruct.buflng;
						FRM_robuf(&FrameReleaseOutputBufferStruct); 	/* release output buffer */

						Error = 3; 					/* set error level for FRM_write */

						if (FrameReleaseOutputBufferStruct.status != 0) 		/* check status */
						{
							Error = 4; 				/* set error level for FRM_robuf */
						}
					}
				}
	/*TODO: Fehler auswerten wenn getBuffer fehlschlägt (8071)*/
				PollingStep++;
				timeout = 0;
				break;
			}
/* wait for the answer */
			case 11:
			{
				/* initialize read structure */
				FRM_read(&FrameReadStruct); 						/* read data form interface */

				if (FrameReadStruct.status == 0) 					/* check status */
				{
					/* Checksum ok? */
					USINT tmp = CreateChecksum((USINT *)FrameReadStruct.buffer,FrameReadStruct.buflng-2);
					if( tmp == ((USINT *)FrameReadStruct.buffer)[FrameReadStruct.buflng-1] )
					{
						/* checksum OK */
						if(ParseAnswer((USINT *)FrameReadStruct.buffer, THERMO_ADDRESS,
						            FrameReadStruct.buflng, ON_OFF_ARRAY, &testval) != 0)
						{
							Error = 12; /* answer not correct*/
						}
						else	/* Answer formal OK */
						{
							/* Answer formal OK, values in Cooler struct */
						}

					}
					else
					{
						/* checksum error */
						Error = 11;
					}

					/* initialize release buffer structure */
					FrameReleaseBufferStruct.buffer = FrameReadStruct.buffer;	/* get adress of read buffer */
					FrameReleaseBufferStruct.buflng = FrameReadStruct.buflng; 	/* get length of read buffer */

					FRM_rbuf(&FrameReleaseBufferStruct); 			/* release read buffer */

					if (FrameReleaseBufferStruct.status != 0) 				/* check status */
					{
						Error = 6; 					/* set error level for FRM_rbuf */
					}
					PollingStep = 0;
					ResendCounter = 0;
				}
				else
				{
					Error = 5; 						/* set error level for FRM_read */
					timeout++;
					if (timeout >= 20) /* 20*cyclic (->2s) time no answer */
					{
						if(ResendCounter >= 5) /*5 times tried? -> error*/
						{
							PollingStep = 0;
							ResendCounter = 0;
						}
						else
						{
							ErrorCounter++;
							ResendCounter++;
							PollingStep = 10;
						}
					}
				}
				break;
			}

/*********************************************************************************************/
/*********************************************************************************************/
/*********************************************************************************************/
/*  send the SET Setpoint command */
			case 20:
			{
				FRM_gbuf(&FrameGetBufferStruct); 				/* get send buffer */

				if (FrameGetBufferStruct.status == 0) 			/* check status */
				{
					int length;

					switch (SetCommands[CurrentSetCommand])
					{
						case SET_SETPOINT:
							{tmpval = (INT)(Cooler.NewValues.SetPoint*10.0);break;}
						case SET_LIMIT_LOW:
							{tmpval = (INT)(Cooler.NewValues.LimitLow*10.0);break;}
						case SET_LIMIT_HIGH:
							{tmpval = (INT)(Cooler.NewValues.LimitHigh*10.0);break;}
						case SET_HEAT_P:
							{tmpval = (INT)(Cooler.NewValues.HeatP*10.0);break;}
						case SET_HEAT_I:
							{tmpval = (INT)(Cooler.NewValues.HeatI*100.0);break;}
						case SET_HEAT_D:
							{tmpval = (INT)(Cooler.NewValues.HeatD*10.0);break;}
						case SET_COOL_P:
							{tmpval = (INT)(Cooler.NewValues.CoolP*10.0);break;}
						case SET_COOL_I:
							{tmpval = (INT)(Cooler.NewValues.CoolI*100.0);break;}
						case SET_COOL_D:
							{tmpval = (INT)(Cooler.NewValues.CoolD*10.0);break;}
					}
					length = CreateCommand((USINT*)FrameGetBufferStruct.buffer,
					                        THERMO_ADDRESS, SetCommands[CurrentSetCommand], tmpval);
					/* initialize write structure */
					FrameWriteStruct.buffer = FrameGetBufferStruct.buffer;		/* get adress of send buffer */
					FrameWriteStruct.buflng = length;

					FRM_write(&FrameWriteStruct); 				/* write data to interface */

					if (FrameWriteStruct.status != 0) 			/* check status */
					{
						/* initialize release output buffer structure */
						FrameReleaseOutputBufferStruct.buffer = FrameGetBufferStruct.buffer;
						FrameReleaseOutputBufferStruct.buflng = FrameGetBufferStruct.buflng;
						FRM_robuf(&FrameReleaseOutputBufferStruct); 	/* release output buffer */

						Error = 3; 					/* set error level for FRM_write */

						if (FrameReleaseOutputBufferStruct.status != 0) 		/* check status */
						{
							Error = 4; 				/* set error level for FRM_robuf */
						}
					}
				}
	/*TODO: Fehler auswerten wenn getBuffer fehlschlägt (8071)*/
				PollingStep++;
				timeout = 0;
				break;
			}
/* wait for the answer */
			case 21:
			{
				/* initialize read structure */
				FRM_read(&FrameReadStruct); 						/* read data form interface */

				if (FrameReadStruct.status == 0) 					/* check status */
				{
					/* Checksum ok? */
					USINT tmp = CreateChecksum((USINT *)FrameReadStruct.buffer,FrameReadStruct.buflng-2);
					if( tmp == ((USINT *)FrameReadStruct.buffer)[FrameReadStruct.buflng-1] )
					{
						/* checksum OK */
						if(ParseAnswer((USINT *)FrameReadStruct.buffer, THERMO_ADDRESS,
						            FrameReadStruct.buflng, SetCommands[CurrentSetCommand], &testval) != 0)
						{
							Error = 12; /* answer not correct*/
						}
						else	/* Answer formal OK */
						{
							/* Answer formal OK, values in Cooler struct */
							switch (SetCommands[CurrentSetCommand])
							{
								case SET_SETPOINT:
									{Cooler.CurrentValues.SetPoint = testval;break;}
								case SET_LIMIT_LOW:
									{Cooler.CurrentValues.LimitLow = testval;break;}
								case SET_LIMIT_HIGH:
									{Cooler.CurrentValues.LimitHigh = testval;break;}
								case SET_HEAT_P:
									{Cooler.CurrentValues.HeatP = testval;break;}
								case SET_HEAT_I:
									{Cooler.CurrentValues.HeatI = testval;break;}
								case SET_HEAT_D:
									{Cooler.CurrentValues.HeatD = testval;break;}
								case SET_COOL_P:
									{Cooler.CurrentValues.CoolP = testval;break;}
								case SET_COOL_I:
									{Cooler.CurrentValues.CoolI = testval;break;}
								case SET_COOL_D:
									{Cooler.CurrentValues.CoolD = testval;break;}
							}
						}

					}
					else
					{
						/* checksum error */
						Error = 11;
					}

					/* initialize release buffer structure */
					FrameReleaseBufferStruct.buffer = FrameReadStruct.buffer;	/* get adress of read buffer */
					FrameReleaseBufferStruct.buflng = FrameReadStruct.buflng; 	/* get length of read buffer */

					FRM_rbuf(&FrameReleaseBufferStruct); 			/* release read buffer */

					if (FrameReleaseBufferStruct.status != 0) 				/* check status */
					{
						Error = 6; 					/* set error level for FRM_rbuf */
					}
					CurrentReadCommand = 0;
					ResendCounter = 0;
					if (CurrentSetCommand < 9 && !SetPointOnly)
					{
						CurrentSetCommand++;
						PollingStep = 20;
					}
					else
					{
						CurrentSetCommand = 0;
						PollingStep = 1;
					}
				}
				else
				{
					Error = 5; 						/* set error level for FRM_read */
					timeout++;
					if (timeout >= 20) /* 20*cyclic (->2s) time no answer */
					{
						if(ResendCounter >= 5) /*5 times tried? -> error*/
						{
							if (CurrentSetCommand < 9)
							{
								CurrentSetCommand++;
								PollingStep = 20;
							}
							else
							{
								CurrentSetCommand = 0;
								PollingStep = 0;
							}
							ResendCounter = 0;
						}
						else
						{
							ErrorCounter++;
							ResendCounter++;
							PollingStep = 20;
						}
					}
				}
				break;
			}

		} /*switch*/
	}
}
```

### Program Logical/Processor/tanks (ANSIC, version 1.12.0) - prewash, rinse and gum tank functions

#### prewash.c
```c
#ifdef _DEFAULT_INCLUDES
	#include <AsDefault.h>
#endif
/*
                             *******************
******************************* C SOURCE FILE *******************************
**                           *******************                           **
**                                                                         **
** project  : BlueFin                                                      **
** filename : PREWASH.C                                                    **
** version  : 1.11                                                         **
** date     : 20.11.2007                                                   **
**                                                                         **
*****************************************************************************
** Abstract                                                                **
** ========                                                                **
** Handling of prewash functions: Circulation, refill, replenishing,       **
** monitoring Level and (optional) circulation switch                      **
**                                                                         **
** Copyright (c) 2007, Krause-Biagosch GmbH                                **
** All rights reserved.                                                    **
**                                                                         **
*****************************************************************************
VERSION HISTORY:
----------------
Version     : 1.00
Date        : 06.03.2007
Revised by  : Herbert Aden
Description : Original version, moved functionality from
              developertank task to here.

Version     : 1.10
Date        : 03.05.2007
Revised by  : Herbert Aden
Description : added delay for Level not ok error and delays for
              level switch on and off signal

Version     : 1.11
Date        : 20.11.2007
Revised by  : Herbert Aden
Description : added flow control functionality in mode "freshwater only",
              requires the sensor to be mounted in the inflow tube
*/
#define _PREWASH_C_SRC

/****************************************************************************/
/**                                                                        **/
/**                           INCLUDE FILES                                **/
/**                                                                        **/
/****************************************************************************/
#include "egmglob_var.h"

/****************************************************************************/
/**                                                                        **/
/**                       DEFINITIONS AND MACROS                           **/
/**                                                                        **/
/****************************************************************************/
/* NONE */

/****************************************************************************/
/**                                                                        **/
/**                      TYPEDEFS AND STRUCTURES                           **/
/**                                                                        **/
/****************************************************************************/
/* NONE */

/****************************************************************************/
/**                                                                        **/
/**                      PROTOTYPES OF LOCAL FUNCTIONS                     **/
/**                                                                        **/
/****************************************************************************/
/* NONE */

/****************************************************************************/
/**                                                                        **/
/**                      EXPORTED VARIABLES                                **/
/**                                                                        **/
/****************************************************************************/
/* NONE */

/****************************************************************************/
/**                                                                        **/
/**                           GLOBAL VARIABLES                             **/
/**                                                                        **/
/****************************************************************************/
/*NONE*/

/****************************************************************************/
/**                                                                        **/
/**                      TASK-LOCAL VARIABLES                              **/
/**                                                                        **/
/****************************************************************************/
_LOCAL    UINT                PrewashValveTime,PrewashValveTimeToGo;

/****************************************************************************/
/**                                                                        **/
/**                    MODULE-LOCAL VARIABLES                              **/
/**                                                                        **/
/****************************************************************************/
static    TP_10ms_typ         PrewashReplenishmentValveTimer;

static    TON_10ms_typ        PrewashLevelOKTimer,PrewashLevelNOTOKTimer,
                              PrewashLevelErrorTimer,
                              PrewashPumpStartTimer,
                              PrewashFlowDelay,
                              PrewashRefillTimer,
                              PrewashPumpOffTimer,
                              RefillValveSafetyTimer;

static    R_TRIGtyp           PrewashPumpCmdR,
                              PrewashValveCmdR,
                              LevelOKR,
                              LevelNOTOKR;
static    F_TRIGtyp           PrewashValveCmdF;

static    BOOL                PrewashRefillActive;
static    UINT                TmpValveTimePrewash;

/****************************************************************************/
/**                                                                        **/
/**                      EXTERNAL VARIABLES                                **/
/**                                                                        **/
/****************************************************************************/
extern BOOL	Pulse_1s;

/****************************************************************************/
/**                                                                        **/
/**                          EXPORTED FUNCTIONS                            **/
/**                                                                        **/
/****************************************************************************/
void Prewash(void);

/******************************************************************************/
void Prewash(void)
{
/*Level*/
	PrewashLevelOKTimer.IN = EGMPrewash.TankFull;
	PrewashLevelOKTimer.PT = 500; /*5 sec*/
	TON_10ms(&PrewashLevelOKTimer);

	PrewashLevelNOTOKTimer.IN = !EGMPrewash.TankFull;
	PrewashLevelNOTOKTimer.PT = 500; /*5 sec*/
	TON_10ms(&PrewashLevelNOTOKTimer);

	LevelOKR.CLK = PrewashLevelOKTimer.Q;
	LevelNOTOKR.CLK = PrewashLevelNOTOKTimer.Q;
	R_TRIG(&LevelOKR);
	R_TRIG(&LevelNOTOKR);
	if(LevelOKR.Q)
		EGMPrewash.LevelNotInRange = FALSE;
	if(LevelNOTOKR.Q)
		EGMPrewash.LevelNotInRange = TRUE;

/* Fehlermeldung verzögern, erst wird automatisch befüllt */
	PrewashLevelErrorTimer.IN = EGMPrewash.LevelNotInRange;
	PrewashLevelErrorTimer.PT = 2000; /* 20 s */
	TON_10ms(&PrewashLevelErrorTimer);
	EGM_AlarmBitField[3] = (ModulStatus_DI == 1) && PrewashLevelErrorTimer.Q && (EGMPrewashParam.ReplenishingMode != FRESHWATERONLY);

/* REPLENISHING Prewash*/
/* a) per plate*/
	if (Pulse_1s &&(CurrentState == S_PROCESSING)&& (EGMPrewashParam.ReplenishingMode == REPLPERPLATE))
	{
		TmpValveTimePrewash =
				((PrewashReplenishmentPlateCounter * EGMPrewashParam.ReplenishmentPerPlate) / EGMPrewashParam.PumpMlPerSec)*100;
		if (TmpValveTimePrewash >= EGMPrewashParam.MinPumpOnTime)
		{
			PrewashReplenishmentValveTimer.IN = 1;
			PrewashReplenishmentPlateCounter = 0;
		}
	}

/* b) per area*/
	if (Pulse_1s &&(CurrentState == S_PROCESSING)&& (EGMPrewashParam.ReplenishingMode == REPLPERSQM))
	{
		TmpValveTimePrewash =
				((PrewashReplenishmentSqmCounter * EGMPrewashParam.ReplenishmentPerSqm) / EGMPrewashParam.PumpMlPerSec)*100;
		if (TmpValveTimePrewash >= EGMPrewashParam.MinPumpOnTime)
		{
			PrewashReplenishmentValveTimer.IN = 1;
			PrewashReplenishmentSqmCounter = 0;
		}
	}

	if (EGMPrewash.Valve != OPEN )
		PrewashValveTime = TmpValveTimePrewash;

	if (PrewashReplenishmentValveTimer.IN && (EGMPrewash.Valve != OPEN ))
		PrewashReplenishmentValveTimer.PT = PrewashValveTime;

	if (EGMPrewash.Valve == OPEN )
		PrewashValveTimeToGo = PrewashReplenishmentValveTimer.PT - PrewashReplenishmentValveTimer.ET;
	else
		PrewashValveTimeToGo = 0;

	TP_10ms(&PrewashReplenishmentValveTimer);
	PrewashReplenishmentValveTimer.IN = 0;

	PrewashValveCmdR.CLK = PrewashReplenishmentValveTimer.Q;
	R_TRIG(&PrewashValveCmdR);
	if (PrewashValveCmdR.Q && (EGMPrewashParam.ReplenishingMode != FRESHWATERONLY))
		EGMPrewash.Valve = OPEN;

/* Ventil zu nach Zeit oder wenn kein Automatik Modus*/
	PrewashValveCmdF.CLK = PrewashReplenishmentValveTimer.Q && EGMPrewash.Auto;
	F_TRIG(&PrewashValveCmdF);
	if ((PrewashValveCmdF.Q && (EGMPrewashParam.ReplenishingMode != FRESHWATERONLY)) || !ControlVoltageOk)
	{
		EGMPrewash.Valve = CLOSE;
	}

/*Refill Prewash*/
	TON_10ms(&PrewashRefillTimer);

/* automatisch befüllen nur, wenn nicht ausschliesslich Frischwasser verwendet wird*/
	if (EGMPrewashParam.ReplenishingMode != FRESHWATERONLY)
	{
		PrewashRefillTimer.IN = !EGMPrewash.LevelNotInRange;
		PrewashRefillTimer.PT = 200;
/* Füllen nur wenn Automatik modus*/
		if (EGMPrewash.LevelNotInRange && ControlVoltageOk && EGMPrewash.Auto)
		{
			EGMPrewash.Valve = OPEN;
			PrewashRefillActive = TRUE;
		}
		if ((PrewashRefillTimer.Q || !EGMPrewash.Auto) && PrewashRefillActive)
		{
			PrewashRefillActive = FALSE;
			EGMPrewash.Valve = CLOSE;
		}
	}
	else
	{
		PrewashRefillTimer.IN = 0;
		PrewashRefillActive = FALSE;
	}

/*
 * safety: if Valve is open and Tank full indicated close the valve after 10 sec
 */
	RefillValveSafetyTimer.IN = (EGMPrewash.Valve == OPEN) && EGMPrewash.TankFull;
	RefillValveSafetyTimer.PT = 1000; /* 10 sec */
	TON_10ms(&RefillValveSafetyTimer);

	if(RefillValveSafetyTimer.Q)
		EGMPrewash.Valve = CLOSE;

	PrewashPumpCmdR.CLK = EGMPrewash.PumpCmd;
	R_TRIG(&PrewashPumpCmdR);

/****************************************************************************/
/**                          Flow control                                  **/
/****************************************************************************/
	if(	EGMGlobalParam.UsePrewashFlowControl )
	{
	/*
	 * wenn ausschliesslich Frischwasser verwendet wird,
	 * dann darf flow control nur  auf das geöffnete Ventil reagieren
	 */
		if (EGMPrewashParam.ReplenishingMode == FRESHWATERONLY)
		{
		/*
		 * 20 sec nach Öffnen muss Durchfluß da sein
		 */
			PrewashPumpStartTimer.IN = EGMPrewash.Valve;
			PrewashPumpStartTimer.PT = 2000; /* 20 sec */
			TON_10ms(&PrewashPumpStartTimer);
			if( PrewashPumpStartTimer.Q && !PrewashFlowInput )
				EGM_AlarmBitField[35] = TRUE;
		}
		else
		{
	/*
	 * 20 sec nach Start der Pumpe muss Durchfluß da sein
	 */
			PrewashPumpStartTimer.IN = EGMPrewash.Pump;
			PrewashPumpStartTimer.PT = 2000; /* 20 sec */
			TON_10ms(&PrewashPumpStartTimer);
	/*
	 * wenn Frischwasser zugeführt wird, schaltet der Durchflußwächter ab,
	 * deshalb hier die Verriegelung des Fehlers mit dem Ventil
	 */
			PrewashFlowDelay.IN = !PrewashFlowInput && !EGMPrewash.Valve;
			PrewashFlowDelay.PT = 300; /* 3 sec */
			TON_10ms(&PrewashFlowDelay);
			if( PrewashPumpStartTimer.Q && PrewashFlowDelay.Q )
				EGM_AlarmBitField[35] = TRUE;
		}
	}
	else
		EGM_AlarmBitField[35] = FALSE;

/* Prewash Pump
 * wenn 30 sec der Level nicht ok war wird die Pumpe abgeschaltet.
 * Sie kann durch steigende Flanke des Kommandos wieder für 30 s eingeschaltet werden
 * (für Service)
*/
	PrewashPumpOffTimer.IN = EGMPrewash.LevelNotInRange && !PrewashPumpCmdR.Q;
	PrewashPumpOffTimer.PT = 3000; /*30 sec*/
	TON_10ms(&PrewashPumpOffTimer);
	if (PrewashPumpOffTimer.Q || !ControlVoltageOk || EGM_AlarmBitField[35])
	{
		EGMPrewash.Pump = OFF;
		EGMPrewash.PumpCmd = OFF;
	}
	else
		EGMPrewash.Pump = EGMPrewash.PumpCmd;

}
/****************************************************************************/
/**                                                                        **/
/**                                 EOF                                    **/
/**                                                                        **/
/****************************************************************************/
```
